{attribute addProperty BoxType "EL3423-0000-0016"}
{attribute addProperty Id "Active_Power_AvgAT %I*REAL32417Active_Power_MinAT %I*REAL32418Active_Power_MaxAT %I*REAL32419Apparent_Power_AvgAT %I*REAL32420Apparent_Power_MinAT %I*REAL32421Apparent_Power_MaxAT %I*REAL32422Reactive_Power_AvgAT %I*REAL32423Reactive_Power_MinAT %I*REAL32424Reactive_Power_MaxAT %I*REAL32425"}
{attribute addProperty CRC "2722643863"}
{attribute addProperty SizeInBites "288"}
{attribute addProperty SizeInBytes "36"}
TYPE Total_Statistic_Power_A2483F97 :
STRUCT
	{attribute addProperty Name "Active_Power_Avg"}
	Active_Power_Avg AT %I* : REAL;
	{attribute addProperty Name "Active_Power_Min"}
	Active_Power_Min AT %I* : REAL;
	{attribute addProperty Name "Active_Power_Max"}
	Active_Power_Max AT %I* : REAL;
	{attribute addProperty Name "Apparent_Power_Avg"}
	Apparent_Power_Avg AT %I* : REAL;
	{attribute addProperty Name "Apparent_Power_Min"}
	Apparent_Power_Min AT %I* : REAL;
	{attribute addProperty Name "Apparent_Power_Max"}
	Apparent_Power_Max AT %I* : REAL;
	{attribute addProperty Name "Reactive_Power_Avg"}
	Reactive_Power_Avg AT %I* : REAL;
	{attribute addProperty Name "Reactive_Power_Min"}
	Reactive_Power_Min AT %I* : REAL;
	{attribute addProperty Name "Reactive_Power_Max"}
	Reactive_Power_Max AT %I* : REAL;
END_STRUCT
END_TYPE

(* stored: Version 1.2.0.0, ProductVersion 3.1.4024.9
   DUT Total_Statistic_Power_A2483F97: Id {4ebbecdb-51d7-44ea-b74f-62d6a014b08a} *)
